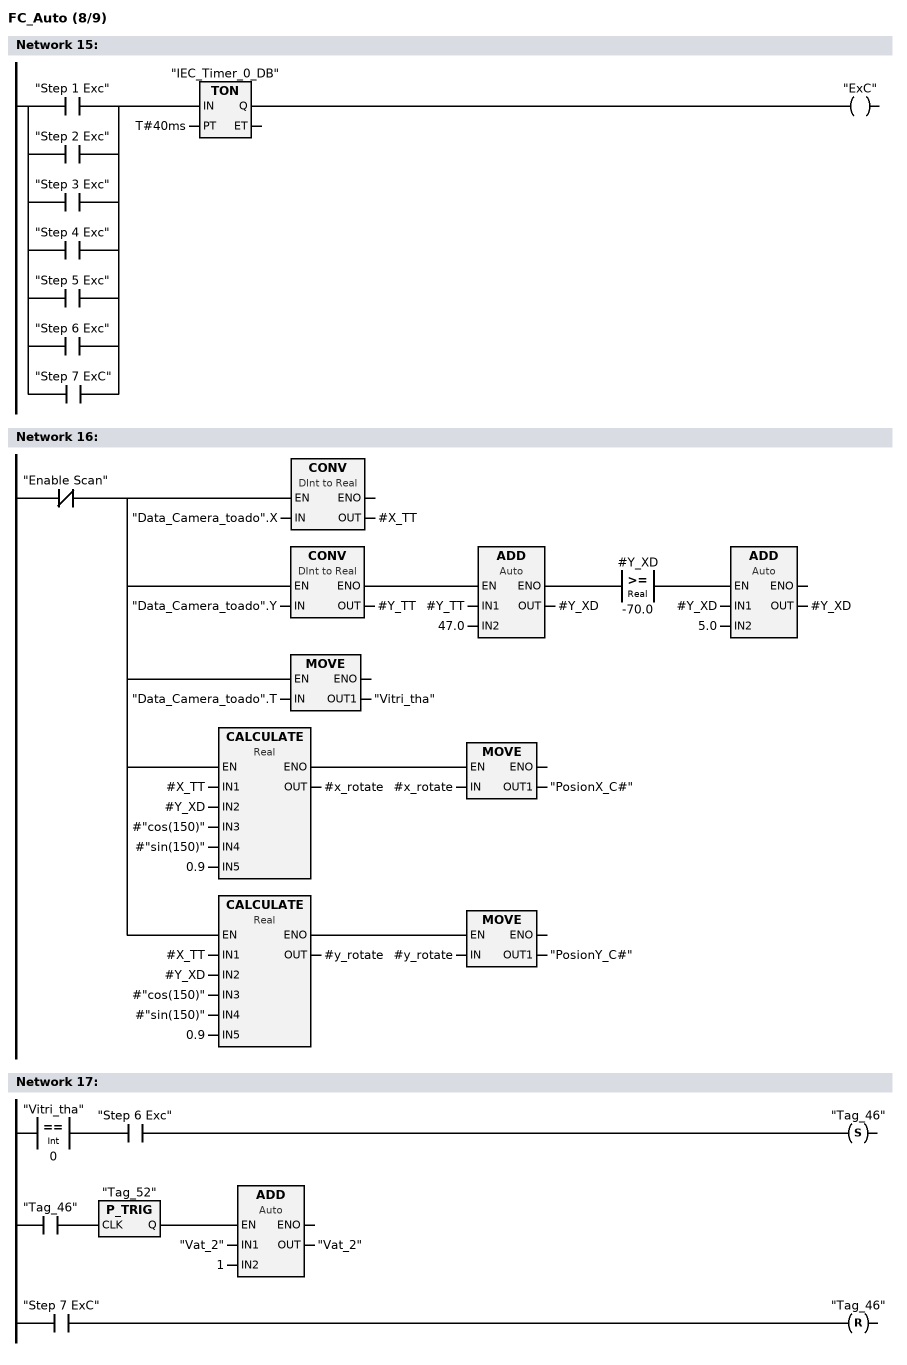
   "IEC_Timer_0_DB".TON(IN := "Step 1 Exc" OR "Step 2 Exc" OR "Step 3 Exc" OR "Step 4 Exc" OR "Step 5 Exc" OR "Step 6 Exc" OR "Step 7 ExC",
                        PT := T#40ms);
   "ExC" := "IEC_Timer_0_DB".Q;
END_REGION

REGION Network 16
   RUNG wire#powerrail
      I_Contact( "Enable Scan" )
      wire#w1
      { S7_Templates := "[SrcType := DInt, DestType := Real]" } Convert(in := "Data_Camera_toado".X, out => #X_TT)
   END_RUNG
   RUNG wire#w1
      { S7_Templates := "[SrcType := DInt, DestType := Real]" } Convert(in := "Data_Camera_toado".Y, out => #Y_TT)
      Add(in1 := #Y_TT, in2 := 47.0, out => #Y_XD)
      { S7_Templates := "SrcType := Real" } GE_Contact(in1 := #Y_XD, in2 := -70.0)
      Add(in1 := #Y_XD, in2 := 5.0, out => #Y_XD)
   END_RUNG
   RUNG wire#w1
      Move(in := "Data_Camera_toado".T, out1 => "Vitri_tha")
   END_RUNG
   RUNG wire#w1
      { S7_Templates := "SrcType := Real"; S7_Expression := "((IN1/IN5*IN3)-(IN4*IN2/IN5))" } Calculate(in1 := #X_TT, in2 := #Y_XD, in3 := #"cos(150)", in4 := #"sin(150)", in5 := 0.9, out => #x_rotate)
      Move(in := #x_rotate, out1 => "PosionX_C#")
   END_RUNG
   RUNG wire#w1
      { S7_Templates := "SrcType := Real"; S7_Expression := "((IN1/IN5*IN4)+(IN2/IN5*IN3))" } Calculate(in1 := #X_TT, in2 := #Y_XD, in3 := #"cos(150)", in4 := #"sin(150)", in5 := 0.9, out => #y_rotate)
      Move(in := #y_rotate, out1 => "PosionY_C#")
   END_RUNG
   // the same network as SCL:
   IF NOT "Enable Scan" THEN
       #X_TT := DINT_TO_REAL("Data_Camera_toado".X);
       #Y_TT := DINT_TO_REAL("Data_Camera_toado".Y);
       #Y_XD := #Y_TT + 47.0;
   END_IF;
   IF NOT "Enable Scan" AND (#Y_XD >= (-70.0)) THEN #Y_XD := #Y_XD + 5.0; END_IF;
   IF NOT "Enable Scan" THEN
       "Vitri_tha" := "Data_Camera_toado".T;
       #x_rotate := ((#X_TT/0.9*#"cos(150)")-(#"sin(150)"*#Y_XD/0.9));
       "PosionX_C#" := #x_rotate;
       #y_rotate := ((#X_TT/0.9*#"sin(150)")+(#Y_XD/0.9*#"cos(150)"));
       "PosionY_C#" := #y_rotate;
   END_IF;
END_REGION

REGION Network 17
   RUNG wire#powerrail
      { S7_Templates := "SrcType := Int" } EQ_Contact(in1 := "Vitri_tha", in2 := 0)
      Contact( "Step 6 Exc" )
      S_Coil( "Tag_46" )
   END_RUNG
   RUNG wire#powerrail
      Contact( "Tag_46" )
      P_Trig( "Tag_52" )
      Add(in1 := "Vat_2", in2 := 1, out => "Vat_2")
   END_RUNG
   RUNG wire#powerrail
      Contact( "Step 7 ExC" )
      R_Coil( "Tag_46" )
   END_RUNG
   // the same network as SCL:
   IF ("Vitri_tha" = 0) AND "Step 6 Exc" THEN "Tag_46" := TRUE; END_IF;
   #_w1 := "Tag_46" AND NOT "Tag_52";   // rising edge
   "Tag_52" := "Tag_46";
   IF #_w1 THEN "Vat_2" := "Vat_2" + 1; END_IF;
   IF "Step 7 ExC" THEN "Tag_46" := FALSE; END_IF;
END_REGION

REGION Network 18
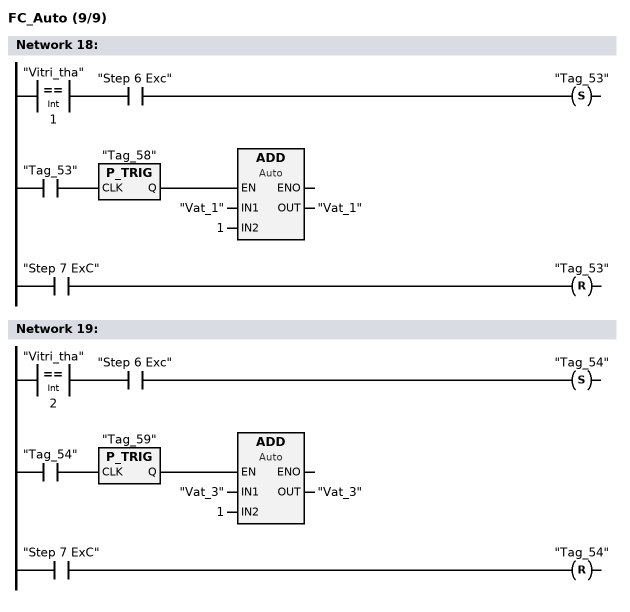
   RUNG wire#powerrail
      { S7_Templates := "SrcType := Int" } EQ_Contact(in1 := "Vitri_tha", in2 := 1)
      Contact( "Step 6 Exc" )
      S_Coil( "Tag_53" )
   END_RUNG
   RUNG wire#powerrail
      Contact( "Tag_53" )
      P_Trig( "Tag_58" )
      Add(in1 := "Vat_1", in2 := 1, out => "Vat_1")
   END_RUNG
   RUNG wire#powerrail
      Contact( "Step 7 ExC" )
      R_Coil( "Tag_53" )
   END_RUNG
   // the same network as SCL:
   IF ("Vitri_tha" = 1) AND "Step 6 Exc" THEN "Tag_53" := TRUE; END_IF;
   #_w1 := "Tag_53" AND NOT "Tag_58";   // rising edge
   "Tag_58" := "Tag_53";
   IF #_w1 THEN "Vat_1" := "Vat_1" + 1; END_IF;
   IF "Step 7 ExC" THEN "Tag_53" := FALSE; END_IF;
END_REGION

REGION Network 19
   RUNG wire#powerrail
      { S7_Templates := "SrcType := Int" } EQ_Contact(in1 := "Vitri_tha", in2 := 2)
      Contact( "Step 6 Exc" )
      S_Coil( "Tag_54" )
   END_RUNG
   RUNG wire#powerrail
      Contact( "Tag_54" )
      P_Trig( "Tag_59" )
      Add(in1 := "Vat_3", in2 := 1, out => "Vat_3")
   END_RUNG
   RUNG wire#powerrail
      Contact( "Step 7 ExC" )
      R_Coil( "Tag_54" )
   END_RUNG
   // the same network as SCL:
   IF ("Vitri_tha" = 2) AND "Step 6 Exc" THEN "Tag_54" := TRUE; END_IF;
   #_w1 := "Tag_54" AND NOT "Tag_59";   // rising edge
   "Tag_59" := "Tag_54";
   IF #_w1 THEN "Vat_3" := "Vat_3" + 1; END_IF;
   IF "Step 7 ExC" THEN "Tag_54" := FALSE; END_IF;
END_REGION
END_FUNCTION

FUNCTION "Fc_soluong_vat" : Void   // FC15, LAD
{ S7_Optimized_Access := 'TRUE' }
VERSION : 0.1
   VAR_TEMP
      v1 : Real;
      v2 : Real;
      v3 : Real;
   END_VAR
BEGIN

REGION Network 1
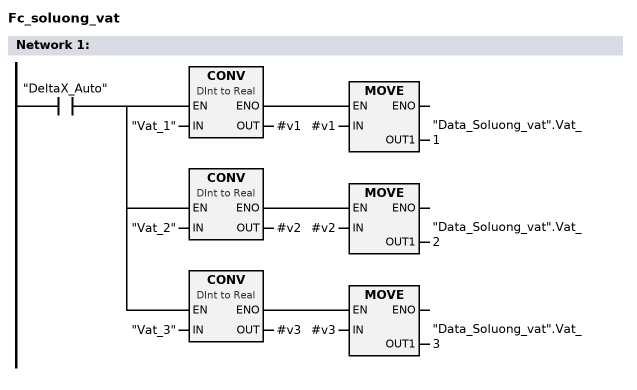
   RUNG wire#powerrail
      Contact( "DeltaX_Auto" )
      wire#w1
      { S7_Templates := "[SrcType := DInt, DestType := Real]" } Convert(in := "Vat_1", out => #v1)
      Move(in := #v1, out1 => "Data_Soluong_vat".Vat_1)
   END_RUNG
   RUNG wire#w1
      { S7_Templates := "[SrcType := DInt, DestType := Real]" } Convert(in := "Vat_2", out => #v2)
      Move(in := #v2, out1 => "Data_Soluong_vat".Vat_2)
   END_RUNG
   RUNG wire#w1
      { S7_Templates := "[SrcType := DInt, DestType := Real]" } Convert(in := "Vat_3", out => #v3)
      Move(in := #v3, out1 => "Data_Soluong_vat".Vat_3)
   END_RUNG
   // the same network as SCL:
   IF "DeltaX_Auto" THEN
       #v1 := DINT_TO_REAL("Vat_1");
       "Data_Soluong_vat".Vat_1 := #v1;
       #v2 := DINT_TO_REAL("Vat_2");
       "Data_Soluong_vat".Vat_2 := #v2;
       #v3 := DINT_TO_REAL("Vat_3");
       "Data_Soluong_vat".Vat_3 := #v3;
   END_IF;
END_REGION
END_FUNCTION

FUNCTION "Button Start" : Void   // FC16, LAD
{ S7_Optimized_Access := 'TRUE' }
VERSION : 0.1
BEGIN

REGION Network 1
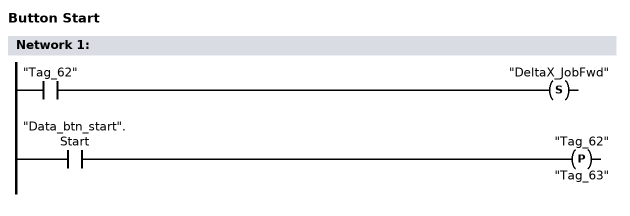
   IF "Tag_62" THEN "DeltaX_JobFwd" := TRUE; END_IF;
   "Tag_62" := "Data_btn_start".Start AND NOT "Tag_63";   // rising edge
   "Tag_63" := "Data_btn_start".Start;
END_REGION
END_FUNCTION

FUNCTION "Button Manual" : Void   // FC17, LAD
{ S7_Optimized_Access := 'TRUE' }
VERSION : 0.1
BEGIN

REGION Network 1
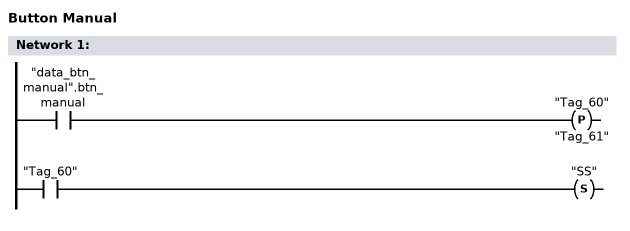
   "Tag_60" := "data_btn_manual".btn_manual AND NOT "Tag_61";   // rising edge
   "Tag_61" := "data_btn_manual".btn_manual;
   IF "Tag_60" THEN "SS" := TRUE; END_IF;
END_REGION
END_FUNCTION

ORGANIZATION_BLOCK "Main"   // OB1, LAD, ProgramCycle
TITLE = "Main Program Sweep (Cycle)"
{ S7_Optimized_Access := 'TRUE' }
VERSION : 0.1
   VAR_INPUT
      Initial_Call : Bool;   // Initial call of this OB
      Remanence : Bool;   // =True, if remanent data are available
   END_VAR
   VAR_TEMP
      theta_1 : Real;
      theta_2 : Real;
      theta_3 : Real;
   END_VAR
   VAR_TEMP   // added for the SCL form of the ladder/FBD networks
      _w1 : Bool;
      _w2 : Bool;
   END_VAR
BEGIN

REGION Network 1
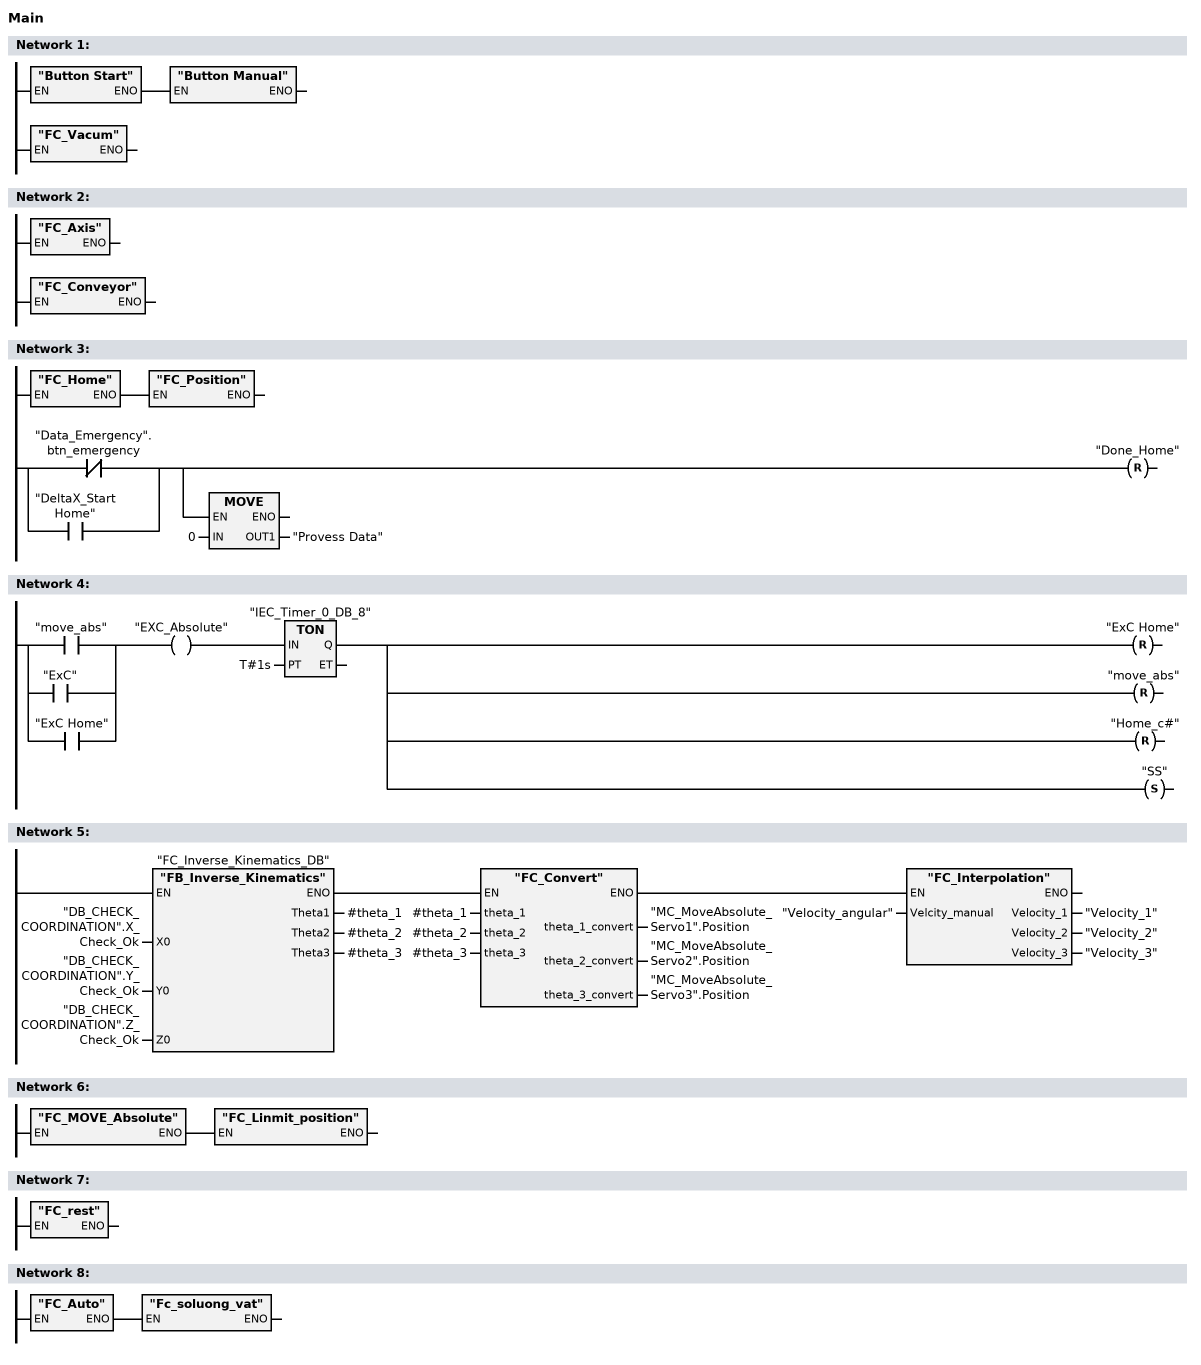
   RUNG wire#powerrail
      "Button Start"()
      "Button Manual"()
   END_RUNG
   RUNG wire#powerrail
      "FC_Vacum"()
   END_RUNG
   // the same network as SCL:
   "Button Start"(ENO => #_w1);
   IF #_w1 THEN "Button Manual"(); END_IF;
   "FC_Vacum"();
END_REGION

REGION Network 2
   RUNG wire#powerrail
      "FC_Axis"()
   END_RUNG
   RUNG wire#powerrail
      "FC_Conveyor"()
   END_RUNG
   // the same network as SCL:
   "FC_Axis"();
   "FC_Conveyor"();
END_REGION

REGION Network 3
   RUNG wire#powerrail
      "FC_Home"()
      "FC_Position"()
   END_RUNG
   RUNG wire#powerrail
      I_Contact( "Data_Emergency".btn_emergency )
      wire#w1
      R_Coil( "Done_Home" )
   END_RUNG
   RUNG wire#powerrail
      Contact( "DeltaX_Start Home" )
   END_RUNG wire#w1
   RUNG wire#w1
      Move(in := 0, out1 => "Provess Data")
   END_RUNG
   // the same network as SCL:
   "FC_Home"(ENO => #_w1);
   IF #_w1 THEN "FC_Position"(); END_IF;
   IF NOT "Data_Emergency".btn_emergency OR "DeltaX_Start Home" THEN
       "Done_Home" := FALSE;
       "Provess Data" := 0;
   END_IF;
END_REGION

REGION Network 4
   "EXC_Absolute" := "move_abs" OR "ExC" OR "ExC Home";
   "IEC_Timer_0_DB_8".TON(IN := "EXC_Absolute", PT := T#1s);
   IF "IEC_Timer_0_DB_8".Q THEN
       "ExC Home" := FALSE;
       "move_abs" := FALSE;
       "Home_c#" := FALSE;
       "SS" := TRUE;
   END_IF;
END_REGION

REGION Network 5
   RUNG wire#powerrail
      "FC_Inverse_Kinematics_DB"(X0 := "DB_CHECK_COORDINATION".X_Check_Ok, Y0 := "DB_CHECK_COORDINATION".Y_Check_Ok, Z0 := "DB_CHECK_COORDINATION".Z_Check_Ok, Theta1 => #theta_1, Theta2 => #theta_2, Theta3 => #theta_3)
      "FC_Convert"(theta_1 := #theta_1, theta_2 := #theta_2, theta_3 := #theta_3, theta_1_convert => "MC_MoveAbsolute_Servo1".Position, theta_2_convert => "MC_MoveAbsolute_Servo2".Position, theta_3_convert => "MC_MoveAbsolute_Servo3".Position)
      "FC_Interpolation"(Velcity_manual := "Velocity_angular", Velocity_1 => "Velocity_1", Velocity_2 => "Velocity_2", Velocity_3 => "Velocity_3")
   END_RUNG
   // the same network as SCL:
   "FC_Inverse_Kinematics_DB"(X0 := "DB_CHECK_COORDINATION".X_Check_Ok,   // "FB_Inverse_Kinematics"
                           Y0 := "DB_CHECK_COORDINATION".Y_Check_Ok,
                           Z0 := "DB_CHECK_COORDINATION".Z_Check_Ok,
                           Theta1 => #theta_1,
                           Theta2 => #theta_2,
                           Theta3 => #theta_3,
                           ENO => #_w1);
   "FC_Convert"(EN := #_w1,
                theta_1 := #theta_1,
                theta_2 := #theta_2,
                theta_3 := #theta_3,
                theta_1_convert => "MC_MoveAbsolute_Servo1".Position,
                theta_2_convert => "MC_MoveAbsolute_Servo2".Position,
                theta_3_convert => "MC_MoveAbsolute_Servo3".Position,
                ENO => #_w2);
   IF #_w2 THEN
       "FC_Interpolation"(Velcity_manual := "Velocity_angular",
                          Velocity_1 => "Velocity_1",
                          Velocity_2 => "Velocity_2",
                          Velocity_3 => "Velocity_3");
   END_IF;
END_REGION

REGION Network 6
   RUNG wire#powerrail
      "FC_MOVE_Absolute"()
      "FC_Linmit_position"()
   END_RUNG
   // the same network as SCL:
   "FC_MOVE_Absolute"(ENO => #_w1);
   IF #_w1 THEN "FC_Linmit_position"(); END_IF;
END_REGION

REGION Network 7
   RUNG wire#powerrail
      "FC_rest"()
   END_RUNG
   // the same network as SCL:
   "FC_rest"();
END_REGION

REGION Network 8
   RUNG wire#powerrail
      "FC_Auto"()
      "Fc_soluong_vat"()
   END_RUNG
   // the same network as SCL:
   "FC_Auto"(ENO => #_w1);
   IF #_w1 THEN "Fc_soluong_vat"(); END_IF;
END_REGION
END_ORGANIZATION_BLOCK